FUNCTION_BLOCK FB_PlantControl
VAR_INPUT
	
	PI_on : BOOL;
	
	PI_Auto : BOOL;
	PI_Manual : BOOL;
	
	PI_Start : BOOL;
	PI_Stop : BOOL;
	PI_Reset : BOOL;
	PI_EmgStop : BOOL;
	
END_VAR
VAR_OUTPUT
	PO_ON : BOOL;
	
	PO_Auto : BOOL;
	PO_Manual : BOOL;
	
	PO_Startet : BOOL;
	PO_Stopped : BOOL;
	PO_Reset : BOOL;
	PO_ResetEmgStop_5s :BOOL;
	
	PO_EmgStopped : BOOL;
	
	PO_Mode_Control : ENUM_MODE_HANDLER;
	
END_VAR
VAR
	EmgResetTimerOff : Tc2_Standard.TON;
	
END_VAR
VAR_IN_OUT
	
	SCADA_Ctrl_Plant : Udt_PlantControl;
	
END_VAR

VAR CONSTANT
	SR_Auto: SR;
	SR_Man : SR;
	
	SR_start : SR;
	SR_Stop : SR;
	SR_EMGStop: SR;
	
END_VAR

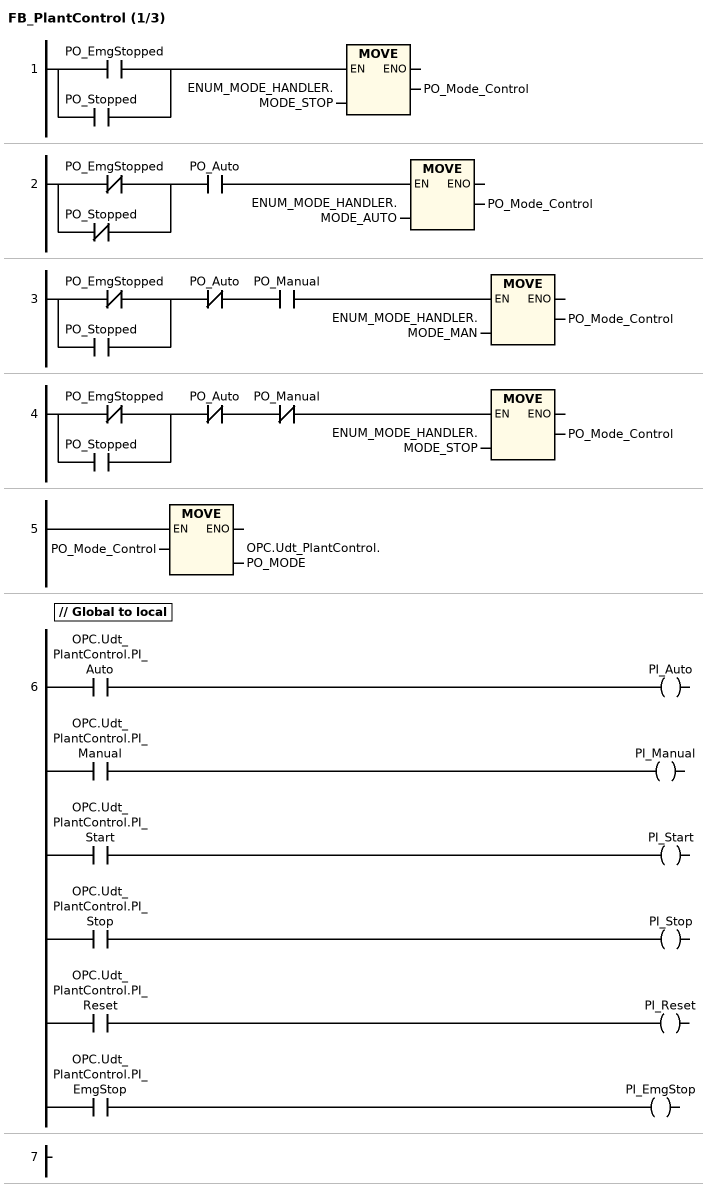
// NETWORK 1
IF PO_EmgStopped OR PO_Stopped THEN PO_Mode_Control := ENUM_MODE_HANDLER.MODE_STOP; END_IF

// NETWORK 2
IF (NOT PO_EmgStopped OR NOT PO_Stopped) AND PO_Auto THEN PO_Mode_Control := ENUM_MODE_HANDLER.MODE_AUTO; END_IF

// NETWORK 3
IF (NOT PO_EmgStopped OR PO_Stopped) AND NOT PO_Auto AND PO_Manual THEN
    PO_Mode_Control := ENUM_MODE_HANDLER.MODE_MAN;
END_IF

// NETWORK 4
IF (NOT PO_EmgStopped OR PO_Stopped) AND NOT PO_Auto AND NOT PO_Manual THEN
    PO_Mode_Control := ENUM_MODE_HANDLER.MODE_STOP;
END_IF

// NETWORK 5
OPC.Udt_PlantControl.PO_MODE := PO_Mode_Control;

// NETWORK 6
// label: // Global to local
PI_Auto := OPC.Udt_PlantControl.PI_Auto;
PI_Manual := OPC.Udt_PlantControl.PI_Manual;
PI_Start := OPC.Udt_PlantControl.PI_Start;
PI_Stop := OPC.Udt_PlantControl.PI_Stop;
PI_Reset := OPC.Udt_PlantControl.PI_Reset;
PI_EmgStop := OPC.Udt_PlantControl.PI_EmgStop;

// NETWORK 7

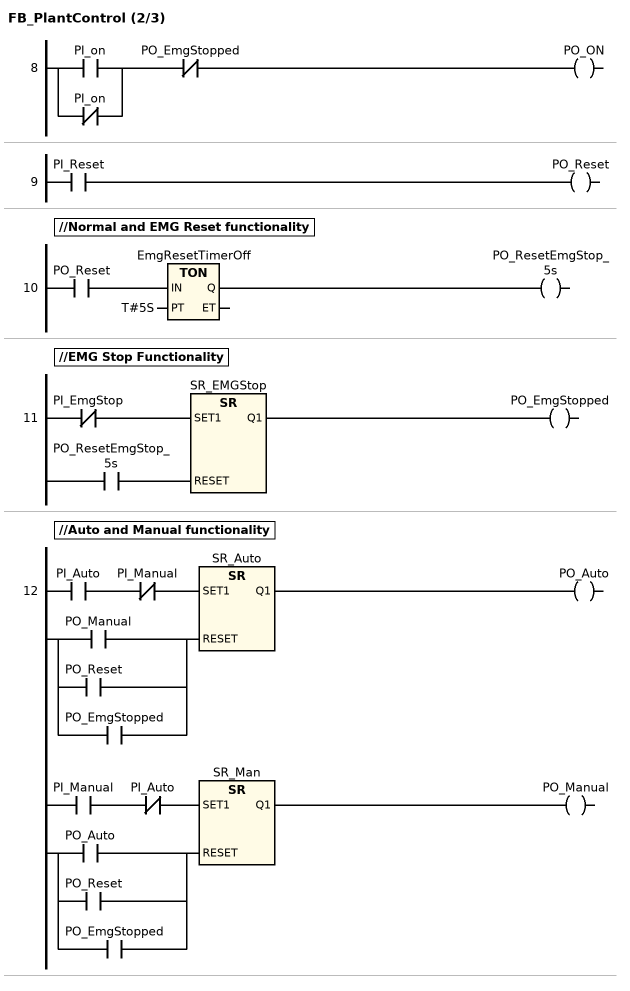
// NETWORK 8
PO_ON := (PI_on OR NOT PI_on) AND NOT PO_EmgStopped;

// NETWORK 9
PO_Reset := PI_Reset;

// NETWORK 10
// label: //Normal and EMG Reset functionality
EmgResetTimerOff(IN := PO_Reset, PT := T#5S); // TON
PO_ResetEmgStop_5s := EmgResetTimerOff.Q;

// NETWORK 11
// label: //EMG Stop Functionality
SR_EMGStop(SET1 := NOT PI_EmgStop, RESET := PO_ResetEmgStop_5s); // SR
PO_EmgStopped := SR_EMGStop.Q1;

// NETWORK 12
// label: //Auto and Manual functionality
SR_Auto(SET1 := PI_Auto AND NOT PI_Manual, RESET := PO_Manual OR PO_Reset OR PO_EmgStopped); // SR
PO_Auto := SR_Auto.Q1;
SR_Man(SET1 := PI_Manual AND NOT PI_Auto, RESET := PO_Auto OR PO_Reset OR PO_EmgStopped); // SR
PO_Manual := SR_Man.Q1;

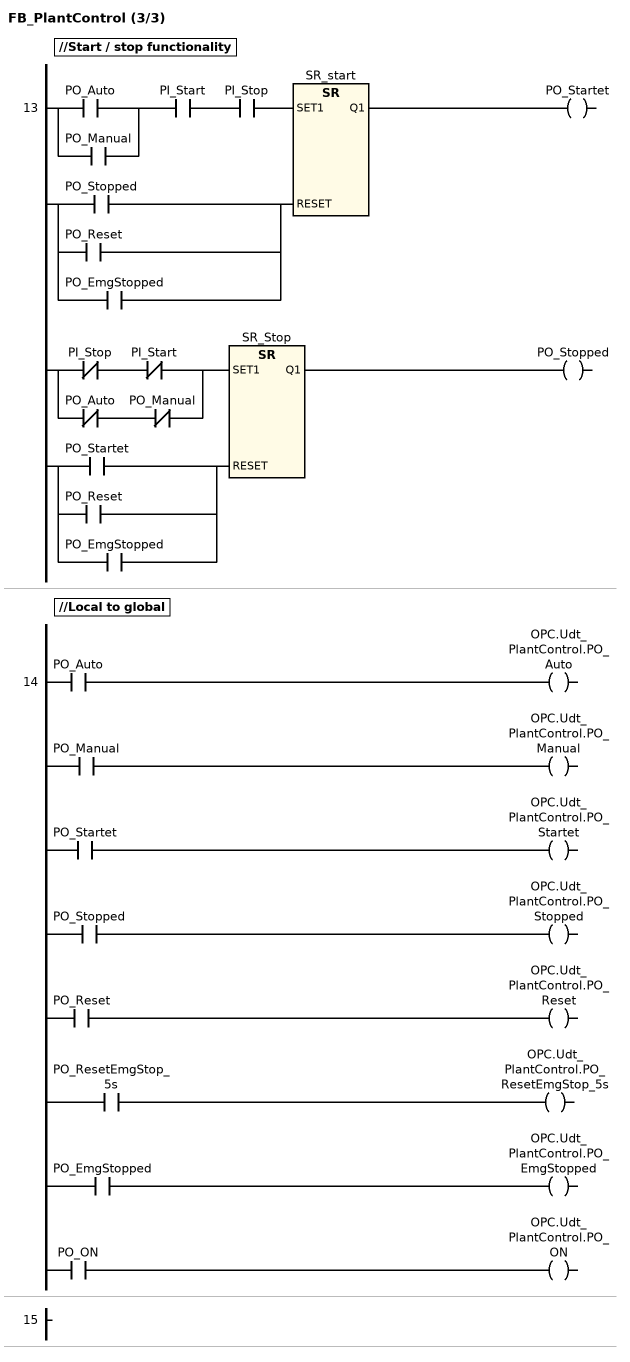
// NETWORK 13
// label: //Start / stop functionality
SR_start(SET1 := (PO_Auto OR PO_Manual) AND PI_Start AND PI_Stop, RESET := PO_Stopped OR PO_Reset OR PO_EmgStopped); // SR
PO_Startet := SR_start.Q1;
SR_Stop(SET1 := NOT PI_Stop AND NOT PI_Start OR NOT PO_Auto AND NOT PO_Manual, RESET := PO_Startet OR PO_Reset OR PO_EmgStopped); // SR
PO_Stopped := SR_Stop.Q1;

// NETWORK 14
// label: //Local to global
OPC.Udt_PlantControl.PO_Auto := PO_Auto;
OPC.Udt_PlantControl.PO_Manual := PO_Manual;
OPC.Udt_PlantControl.PO_Startet := PO_Startet;
OPC.Udt_PlantControl.PO_Stopped := PO_Stopped;
OPC.Udt_PlantControl.PO_Reset := PO_Reset;
OPC.Udt_PlantControl.PO_ResetEmgStop_5s := PO_ResetEmgStop_5s;
OPC.Udt_PlantControl.PO_EmgStopped := PO_EmgStopped;
OPC.Udt_PlantControl.PO_ON := PO_ON;

// NETWORK 15

END_FUNCTION_BLOCK

(* stored: Version 1.1.0.1, ProductVersion 3.1.4024.13
   POU FB_PlantControl: Id {b53adaf6-8506-476c-8298-f670f349374b}, SpecialFunc None *)
